FUNCTION ASCF_CL_36_XNOR : WORD
VAR_OUTPUT
	Out						: ASCF_UnionType;				//Result of the computation (Type: VBool)
END_VAR

VAR_IN_OUT
	Arguments				: ARRAY[0..3] OF ASCF_UnionType;	//Arguments for the function (Arguments: 2 - 4, Type: VBool)
END_VAR

VAR
	tempRet					: WORD;
	constErrors				: ASCF_CL_EnumErrors;				//Enumeration type of the error codes of the Adaptive Logic.
END_VAR



//#################################################################################################
{region "EXECUTE AND OUTPUT"}
    tempRet := ASCF_CL_35_XOR(Arguments := Arguments, Out => Out);
    
    // negate result if XOR was successful
    IF tempRet = constErrors.None THEN
        Out.VBool := NOT Out.VBool;
    END_IF;
    
    ASCF_CL_36_XNOR := tempRet;
{endregion}

END_FUNCTION

(* stored: Version 1.1.0.1, ProductVersion 3.1.4026.4
   POU ASCF_CL_36_XNOR: Id {e0284d83-382e-4fb4-a51a-4f077d3849c1}, SpecialFunc None *)
